// TIA Portal V18 export
TYPE "typeDefectsDB"
// stored: IsFailsafeCompliant false
   STRUCT
      i : Int;
      N : Int;
      N_max : Int := 30;
      pos_AR : Array[1..30] of "typePositions";
   END_STRUCT;
END_TYPE
